PROGRAM Temp
VAR
END_VAR

// NETWORK 1

END_PROGRAM

(* stored: Version 1.1.0.1, ProductVersion 3.1.4024.12
   POU Temp: Id {f4569fdc-e13c-4145-b338-6af60af79f02}, SpecialFunc None *)
